TYPE ST_SL_Zustand :
STRUCT
	Stellung_Anford		: BOOL;
	Stellung_Soll		: BOOL;
	Stellung			: BOOL;

	Freigabe			: BOOL;
	Freigabe_Deakt		: BOOL;
	Freigabe_Code		: WORD;

	Stoerung			: BOOL;
	Stoerung_Code		: WORD;

	Warnung				: BOOL;
	Warnung_Code		: WORD;

	Status				: SINT;

	Stellungwechsel01	: BOOL;
	Stellungwechsel10	: BOOL;

	Quittierung			: BOOL;

END_STRUCT
END_TYPE

(* stored: Version 1.1.0.1, ProductVersion 3.1.4024.9
   DUT ST_SL_Zustand: Id {bdbe1cd7-f7e3-4321-b26d-458b3b7c6c9c} *)
